{attribute 'GeneratedUsingTerminal: EL6861-0000-0016'}
{attribute addProperty BoxType "EL6861-0000-0016"}
{attribute addProperty Id "CtrlAT %Q*Ctrl_E65815995Data_OutAT %Q*ARRAY[0..127] OF USINT128"}
{attribute addProperty CRC "4242093104"}
{attribute addProperty Size "133"}
TYPE COM_RxPDO_Map_01DE24DC EXTENDS OutputBase_10CEE7DE :
STRUCT
	{attribute addProperty Name "Ctrl"}
	Ctrl AT %Q* : Ctrl_E6581599;
	{attribute addProperty Name "Data_Out"}
	Data_Out AT %Q* : ARRAY[0..127] OF USINT;
END_STRUCT
END_TYPE

(* stored: Version 1.2.0.0, ProductVersion 3.1.4024.11
   DUT COM_RxPDO_Map_01DE24DC: Id {760d3532-7a6f-4fac-bf3b-3177a891b20b} *)
